// Mitsubishi GX Works2 project: CNC3Axis   PLC: FX3U/FX3UC

// global labels: Global
VAR_GLOBAL
  IsOn AT M0 : BOOL;
  RunButton AT M1 : BOOL;
  StopButton AT M2 : BOOL;
  ResetButton AT M3 : BOOL;
  SetButton AT M4 : BOOL;
  OriginButton AT M5 : BOOL;
  EmergencyButton AT M6 : BOOL;
  ManualSpeed AT D0 : DINT;
  ManualStepLength AT D2 : DINT;
  StateRun AT D4 : INT;
  StateSetOrigin AT D5 : INT;
  StateMoveToOrigin AT D6 : INT;
  StateFile AT D7 : INT;
  StateBacklash AT D8 : INT;
  OnOffResetStop : OnOffResetStop;
  ManualHandler : ManualHandler;
  AutoHandler : AutoHandler;
  PulseOutAndLimit : PulseOutAndLimit;
  OriginSetMove : OriginSetMove;
  ArrayRun AT M7 : BOOL;
  ArrayIndex AT D9 : DINT;
  ArrayIndexMax AT D11 : DINT;
  ArrayIndexEnd AT D13 : DINT;
  ArrayIndexModulo AT D15 : DINT;
  ArrayData AT D1000 : ARRAY [0..1599] OF INT;
  ArrayStep AT M8 : BOOL;
  ArrayStepManual AT M9 : BOOL;
  XXLimitN AT M8344 : BOOL;
  XXLimitP AT M8343 : BOOL;
  XXBusy AT M8340 : BOOL;
  XXCurPos AT D8340 : DINT;
  XXCurPosView AT D17 : DINT;
  XXTarPos AT D19 : DINT;
  XXCurFS AT D21 : DINT;
  XXToOrigin AT D23 : DINT;
  XXTarR : BOOL;
  XXManualN AT M10 : BOOL;
  XXManualP AT M11 : BOOL;
  XXILimitN AT X010 : BOOL;
  XXILimitP AT X011 : BOOL;
  XXOOnOff AT Y020 : BOOL;
  XXOReset AT Y021 : BOOL;
  XXOPulse AT Y000 : BOOL;
  XXODirection AT Y004 : BOOL;
  XXOEmergencyStop AT Y010 : BOOL;
  XXOBrake AT Y027 : BOOL;
  XXRunLatch : BOOL;
  XXRunLatchFalling : BOOL;
  XXBacklashConstant AT D25 : DINT;
  XXBacklash AT M12 : BOOL;
  XXBacklashDirection AT D27 : INT;
  YYLimitN AT M8354 : BOOL;
  YYLimitP AT M8353 : BOOL;
  YYBusy AT M8350 : BOOL;
  YYCurPos AT D8350 : DINT;
  YYCurPosView AT D28 : DINT;
  YYTarPos AT D30 : DINT;
  YYCurFS AT D32 : DINT;
  YYToOrigin AT D34 : DINT;
  YYTarR : BOOL;
  YYManualN AT M13 : BOOL;
  YYManualP AT M14 : BOOL;
  YYILimitN AT X012 : BOOL;
  YYILimitP AT X013 : BOOL;
  YYOOnOff AT Y022 : BOOL;
  YYOReset AT Y023 : BOOL;
  YYOPulse AT Y001 : BOOL;
  YYODirection AT Y005 : BOOL;
  YYOEmergencyStop AT Y011 : BOOL;
  YYOBrake AT Y031 : BOOL;
  YYRunLatch : BOOL;
  YYRunLatchFalling : BOOL;
  YYBacklashConstant AT D36 : DINT;
  YYBacklash AT M15 : BOOL;
  YYBacklashDirection AT D38 : INT;
  ZZLimitN AT M8364 : BOOL;
  ZZLimitP AT M8363 : BOOL;
  ZZBusy AT M8360 : BOOL;
  ZZCurPos AT D8360 : DINT;
  ZZCurPosView AT D39 : DINT;
  ZZTarPos AT D41 : DINT;
  ZZCurFS AT D43 : DINT;
  ZZToOrigin AT D45 : DINT;
  ZZTarR : BOOL;
  ZZManualN AT M16 : BOOL;
  ZZManualP AT M17 : BOOL;
  ZZILimitN AT X014 : BOOL;
  ZZILimitP AT X015 : BOOL;
  ZZOOnOff AT Y024 : BOOL;
  ZZOReset AT Y025 : BOOL;
  ZZOPulse AT Y002 : BOOL;
  ZZODirection AT Y006 : BOOL;
  ZZOEmergencyStop AT Y012 : BOOL;
  ZZOBrake AT Y033 : BOOL;
  ZZRunLatch : BOOL;
  ZZRunLatchFalling : BOOL;
  ZZBacklashConstant AT D47 : DINT;
  ZZBacklash AT M18 : BOOL;
  ZZBacklashDirection AT D49 : INT;
END_VAR

// task Task_01 (event TRUE, interval 0, priority 31): Main

PROGRAM Main
VAR
  fRising : BOOL;
  fRisingLatch : BOOL;
END_VAR
OnOffResetStop();
IF IsOn THEN
	PLS(RunButton, fRising);
	SET(fRising, fRisingLatch);
	MOV(fRisingLatch AND (StateRun = 0 OR StateRun = 3), 1, StateRun);
	RST(fRisingLatch, fRisingLatch);
	ManualHandler();
	AutoHandler();
	OriginSetMove();
	PulseOutAndLimit();
	XXCurPosView := XXCurPos;
	YYCurPosView := YYCurPos;
	ZZCurPosView := ZZCurPos;
END_IF;
END_PROGRAM

FUNCTION_BLOCK PulseOutAndLimit
VAR
  fRun : BOOL;
  fTarR : BOOL;
  fRising : BOOL;
  fRisingLatch : BOOL;
END_VAR
fRun := StateRun = 2;

(*X Axis ||||||||||||||||||||||||||||||||||||||||*)
OUT(XXILimitN, XXLimitN);
OUT(XXILimitP, XXLimitP);
SET(fRun AND NOT XXTarR, XXRunLatch);
DDRVA(XXRunLatch, XXTarPos, XXCurFS, XXOPulse, XXODirection);
RST(M8029, XXRunLatch);
RST(M8329, XXRunLatch);
PLF(XXRunLatch, XXRunLatchFalling);
SET(XXRunLatchFalling, XXTarR);

(*Y Axis ||||||||||||||||||||||||||||||||||||||||*)
OUT(YYILimitN, YYLimitN);
OUT(YYILimitP, YYLimitP);
SET(fRun AND NOT YYTarR, YYRunLatch);
DDRVA(YYRunLatch, YYTarPos, YYCurFS, YYOPulse, YYODirection);
RST(M8029, YYRunLatch);
RST(M8329, YYRunLatch);
PLF(YYRunLatch, YYRunLatchFalling);
SET(YYRunLatchFalling, YYTarR);

(*Z Axis ||||||||||||||||||||||||||||||||||||||||*)
OUT(ZZILimitN, ZZLimitN);
OUT(ZZILimitP, ZZLimitP);
SET(fRun AND NOT ZZTarR, ZZRunLatch);
DDRVA(ZZRunLatch, ZZTarPos, ZZCurFS, ZZOPulse, ZZODirection);
RST(M8029, ZZRunLatch);
RST(M8329, ZZRunLatch);
PLF(ZZRunLatch, ZZRunLatchFalling);
SET(ZZRunLatchFalling, ZZTarR);

(*Run complete*)
fTarR := fRun AND XXTarR AND YYTarR AND ZZTarR;
RST(fTarR, RunButton);
MOV(fTarR, 3, StateRun);
END_FUNCTION_BLOCK

FUNCTION_BLOCK OnOffResetStop
DMOV(M8002, 1000, ManualSpeed);
DMOV(M8002, 100, ManualStepLength);
DMOV(M8002, 5000, XXToOrigin);
DMOV(M8002, 5000, YYToOrigin);
DMOV(M8002, 5000, ZZToOrigin);
MOV(M8002, 50, D8348);
MOV(M8002, 50, D8349);
MOV(M8002, 50, D8358);
MOV(M8002, 50, D8359);
MOV(M8002, 50, D8368);
MOV(M8002, 50, D8369);

OUT(IsOn, XXOOnOff);
OUT(IsOn, YYOOnOff);
OUT(IsOn, ZZOOnOff);

OUT(EmergencyButton, XXOEmergencyStop);
OUT(EmergencyButton, YYOEmergencyStop);
OUT(EmergencyButton, ZZOEmergencyStop);

OUT(IsOn, XXOBrake);
OUT(IsOn, YYOBrake);
OUT(IsOn, ZZOBrake);

SET(ResetButton, XXOReset);
SET(ResetButton, YYOReset);
SET(ResetButton, ZZOReset);
OUT_T(ResetButton, TC200, 8);
RST(TC200, ResetButton);
RST(TC200, XXOReset);
RST(TC200, YYOReset);
RST(TC200, ZZOReset);

IF StopButton THEN
	RunButton := FALSE;
	XXTarR := FALSE;
	YYTarR := FALSE;
	ZZTarR := FALSE;
	XXRunLatch := FALSE;
	YYRunLatch := FALSE;
	ZZRunLatch := FALSE;
	ArrayRun := FALSE;
	StopButton := FALSE;
	SetButton := FALSE;
	OriginButton := FALSE;
	RST(TRUE, StateRun);
	RST(TRUE, StateSetOrigin);
	RST(TRUE, StateMoveToOrigin);
	RST(TRUE, StateFile);
	RST(TRUE, StateBacklash);
END_IF;
END_FUNCTION_BLOCK

FUNCTION_BLOCK OriginSetMove
VAR
  fReady : BOOL;
  fOriginButtonRising : BOOL;
  fOriginButtonRisingLatch : BOOL;
  fTarR : BOOL;
END_VAR
PLS(OriginButton, fOriginButtonRising);
SET(fOriginButtonRising, fOriginButtonRisingLatch);
fReady := NOT RunButton AND (StateRun = 0 OR StateRun = 3) AND StateBacklash = 0;
fTarR := StateBacklash = 0 AND StateRun = 3 AND NOT XXBusy AND NOT YYBusy AND NOT ZZBusy;

(*Set origin*)
IF fReady AND SetButton AND fOriginButtonRisingLatch THEN
	StateSetOrigin := 1;
	RST(TRUE, StateBacklash);
	XXBacklashDirection := -1;
	YYBacklashDirection := -1;
	ZZBacklashDirection := -1;
	XXTarPos := XXCurPos + (XXToOrigin - 3000);
	YYTarPos := YYCurPos + (YYToOrigin - 3000);
	ZZTarPos := ZZCurPos + (ZZToOrigin - 3000) / 2;
	ManualSpeed := 1000;
	XXCurFS := ManualSpeed;
	YYCurFS := ManualSpeed;
	ZZCurFS := ManualSpeed;
	RunButton := TRUE;
END_IF;

IF StateSetOrigin = 1 THEN
	SET(NOT XXILimitN, XXTarR);
	SET(NOT YYILimitN, YYTarR);
	SET(NOT ZZILimitN, ZZTarR);
	RST(NOT XXILimitN, XXRunLatch);
	RST(NOT YYILimitN, YYRunLatch);
	RST(NOT ZZILimitN, ZZRunLatch);
END_IF;

IF StateSetOrigin = 3 THEN
	RST(TRUE, XXCurPos);
	RST(TRUE, YYCurPos);
	RST(TRUE, ZZCurPos);
	RST(TRUE, XXTarPos);
	RST(TRUE, YYTarPos);
	RST(TRUE, ZZTarPos);
	RST(TRUE, StateSetOrigin);
	RST(TRUE, OriginButton);
	RST(TRUE, SetButton);
END_IF;

MOV(NOT RunButton AND StateSetOrigin = 2 AND fTarR, 3, StateSetOrigin);
MOV(NOT RunButton AND StateSetOrigin = 1 AND fTarR, 2, StateSetOrigin);

(*Move to origin*)
IF fReady AND NOT SetButton AND fOriginButtonRisingLatch THEN
	StateMoveToOrigin := 1;
	XXTarPos := XXCurPos;
	YYTarPos := YYCurPos;
	RST(TRUE, ZZTarPos);
	DMOV(ManualSpeed < 10000, 10000, ManualSpeed);
	XXCurFS := ManualSpeed;
	YYCurFS := ManualSpeed;
	ZZCurFS := ManualSpeed;
	SET(ZZCurPos <> 0, RunButton);
	MOV(NOT RunButton, 3, StateRun);
END_IF;

INC(NOT RunButton AND StateMoveToOrigin > 0 AND fTarR, StateMoveToOrigin);

IF fReady AND StateMoveToOrigin = 2 THEN
	RST(TRUE, XXTarPos);
	RST(TRUE, YYTarPos);
	RunButton := TRUE;
END_IF;

IF StateMoveToOrigin > 2 THEN
	RST(TRUE, StateMoveToOrigin);
	RST(TRUE, OriginButton);
END_IF;

RST(fOriginButtonRisingLatch, fOriginButtonRisingLatch);
END_FUNCTION_BLOCK

FUNCTION_BLOCK ManualHandler
VAR
  fAny : BOOL;
  fAnyX : BOOL;
  fAnyY : BOOL;
  fAnyZ : BOOL;
END_VAR
IF NOT ArrayRun AND (StateRun = 0 OR StateRun = 3) AND StateBacklash = 0 THEN
	fAnyX := XXManualN OR XXManualP;
	fAnyY := YYManualN OR YYManualP;
	fAnyZ := ZZManualN OR ZZManualP;
	fAny := fAnyX OR fAnyY OR fAnyZ;
	DMOV(fAny AND ManualSpeed < 10, 10, ManualSpeed);
	DMOV(fAny AND ManualStepLength < 10, 10, ManualStepLength);
	(**)
	DMOV(fAny, XXCurPos, XXTarPos);
	DSUB(XXManualN, XXTarPos, ManualStepLength, XXTarPos);
	DADD(XXManualP, XXTarPos, ManualStepLength, XXTarPos);
	DMOV(fAny, ManualSpeed, XXCurFS);
	(**)
	DMOV(fAny, YYCurPos, YYTarPos);
	DSUB(YYManualN, YYTarPos, ManualStepLength, YYTarPos);
	DADD(YYManualP, YYTarPos, ManualStepLength, YYTarPos);
	DMOV(fAny, ManualSpeed, YYCurFS);
	(**)
	DMOV(fAny, ZZCurPos, ZZTarPos);
	DSUB(ZZManualN, ZZTarPos, ManualStepLength, ZZTarPos);
	DADD(ZZManualP, ZZTarPos, ManualStepLength, ZZTarPos);
	DMOV(fAny, ManualSpeed, ZZCurFS);
	(**)
	SET(fAny, RunButton);
END_IF;
END_FUNCTION_BLOCK

FUNCTION_BLOCK AutoHandler
VAR
  fTarR : BOOL;
  fArrayRunRising : BOOL;
  fArrayRunRisingLatch : BOOL;
  fArrayRunReady : BOOL;
  fArrayStepRising : BOOL;
  fArrayStepRisingLatch : BOOL;
  fArrayStepReady : BOOL;
  fArrayIndex : DINT;
  fXXTarPos : DINT;
  fYYTarPos : DINT;
  fZZTarPos : DINT;
END_VAR
(*Backlash*)
IF StateRun = 1 AND StateBacklash = 0 THEN
	XXBacklash := XXTarPos <> XXCurPos AND ((XXBacklashDirection < 0 AND XXTarPos > XXCurPos) OR (XXBacklashDirection > 0 AND XXTarPos < XXCurPos));
	YYBacklash := YYTarPos <> YYCurPos AND ((YYBacklashDirection < 0 AND YYTarPos > YYCurPos) OR (YYBacklashDirection > 0 AND YYTarPos < YYCurPos));
	ZZBacklash := ZZTarPos <> ZZCurPos AND ((ZZBacklashDirection < 0 AND ZZTarPos > ZZCurPos) OR (ZZBacklashDirection > 0 AND ZZTarPos < ZZCurPos));
	MOV(XXBacklash, XXBacklashDirection * -1, XXBacklashDirection);
	MOV(YYBacklash, YYBacklashDirection * -1, YYBacklashDirection);
	MOV(ZZBacklash, ZZBacklashDirection * -1, ZZBacklashDirection);
	MOV(XXBacklash OR YYBacklash OR ZZBacklash, 1, StateBacklash);
END_IF;

IF StateRun = 1 AND StateBacklash = 1 THEN
	fXXTarPos := XXTarPos;
	fYYTarPos := YYTarPos;
	fZZTarPos := ZZTarPos;
	DMOV(XXBacklash, XXCurPos + XXBacklashConstant * INT_TO_DINT(XXBacklashDirection), XXTarPos);
	DMOV(YYBacklash, YYCurPos + YYBacklashConstant * INT_TO_DINT(YYBacklashDirection), YYTarPos);
	DMOV(ZZBacklash, ZZCurPos + ZZBacklashConstant * INT_TO_DINT(ZZBacklashDirection), ZZTarPos);
	StateBacklash := 2;
END_IF;

IF StateBacklash = 2 AND (StateRun = 0 OR StateRun = 3) THEN
	DMOV(XXBacklash, XXCurPos - XXBacklashConstant * INT_TO_DINT(XXBacklashDirection), XXCurPos);
	DMOV(YYBacklash, YYCurPos - YYBacklashConstant * INT_TO_DINT(YYBacklashDirection), YYCurPos);
	DMOV(ZZBacklash, ZZCurPos - ZZBacklashConstant * INT_TO_DINT(ZZBacklashDirection), ZZCurPos);
	XXTarPos := fXXTarPos;
	YYTarPos := fYYTarPos;
	ZZTarPos := fZZTarPos;
	RunButton := TRUE;
	StateBacklash := 3;
END_IF;

IF StateBacklash = 3 AND (StateRun = 0 OR StateRun = 3) THEN
	RST(TRUE, StateBacklash);
END_IF;
(*Backlash*)

IF StateRun = 1 THEN
	XXTarR := XXCurPos = XXTarPos;
	YYTarR := YYCurPos = YYTarPos;
	ZZTarR := ZZCurPos = ZZTarPos;
	fTarR := XXTarR AND YYTarR AND ZZTarR;
	RST(fTarR, RunButton);
	MOV(fTarR, 3, StateRun);
	MOV(NOT fTarR, 2, StateRun);
END_IF;

fArrayRunReady := XXCurPos = 0 AND YYCurPos = 0 AND ZZCurPos = 0;
PLS(ArrayRun, fArrayRunRising);
SET(fArrayRunRising, fArrayRunRisingLatch);
MOV(fArrayRunRisingLatch AND fArrayRunReady, 1, StateFile);
RST(fArrayRunRisingLatch AND NOT fArrayRunReady, ArrayRun);
RST(fArrayRunRisingLatch, fArrayRunRisingLatch);
RST(StateFile = 2, ArrayRun);
RST(StateFile = 2, StateFile);

fArrayStepReady := ArrayRun AND (StateRun = 0 OR StateRun = 3) AND StateFile = 1 AND StateBacklash = 0;
PLS(ArrayStep, fArrayStepRising);
SET(fArrayStepRising, fArrayStepRisingLatch);
IF fArrayStepReady AND fArrayStepRisingLatch THEN
	ArrayIndexModulo := ArrayIndex - ((ArrayIndex / 200) * 200);
	fArrayIndex := ArrayIndexModulo * 8;
	MOV(TRUE, DINT_TO_INT(fArrayIndex), Z);
	DMOV(TRUE, D1000Z, XXTarPos);
	DMOV(TRUE, D1002Z, YYTarPos);
	DMOV(TRUE, WORD_TO_DINT(D1004Z), ZZTarPos);
	DMOV(TRUE, WORD_TO_DINT(D1005Z), XXCurFS);
	DMOV(TRUE, WORD_TO_DINT(D1006Z), YYCurFS);
	DMOV(TRUE, WORD_TO_DINT(D1007Z), ZZCurFS);
	SET(TRUE, RunButton);
	MOV(TRUE, 1, StateRun);
	MOV(ArrayIndex = ArrayIndexEnd, 2, StateFile);
	DINC(ArrayIndex < ArrayIndexMax, ArrayIndex);
END_IF;
RST(fArrayStepRisingLatch, ArrayStep);
RST(fArrayStepRisingLatch, fArrayStepRisingLatch);
SET(fArrayStepReady AND ArrayIndexMax > 0 AND NOT ArrayStepManual, fArrayStepRisingLatch);
END_FUNCTION_BLOCK
